(* CoDeSys 2.3 export: FILEHANDLING.EXP *)
(* Libraries: 05_Utilities\MPLCUtilities.lib 30.1.17 00:00:00, 11_System\SysLibFileAsync.lib 27.1.17 13:50:06, 11_System\SysLibProjectInfo.lib 27.1.17 13:50:06, 11_System\SysLibRtc.lib 27.1.17 13:50:06, 12_Additional\Util.lib 27.1.17 13:50:06, Internal\MPLCIntern_Utilities.lib 30.1.17 00:00:00 *)

(* Data type in CodeSamples/FileHandling *)
TYPE ST_CSVData :
STRUCT
	(********************)
	TimeStamp		: STRING(25)	:='                      ';	(* Time stamp *)
	Separator1		: BYTE			:= 16#3B; 			(* Semicolon *)
	Description1		: STRING(25)	:='                         ';	(* Description of the log data *)
	Separator2		: BYTE			:= 16#3B; 			(* Semicolon *)
	Value1				: STRING(25)	:='                         ';	(* Log value *)
	Separator3		: BYTE			:= 16#3B; 			(* Semicolon *)

	(********************)
	Description2		: STRING(25)	:='                         ';	(* Description of the log data *)
	Separato4		: BYTE				:= 16#3B; 			(* Semicolon *)
	Value2				: STRING(25)	:='                         ';	(* Log value *)
	Separator5		: BYTE			:= 16#3B; 			(* Semicolon *)
	GAP			: STRING(2)	:='  '; (*See Description*)
	CRLF3				: WORD		:= 16#0D0A;		(*Carriage return , Line feed*)

	
	(*Attention: 
	  The total number of bytes of the structure must be integer divisible by 4.
	  Use the GAP variable to compensate the size of the structure.
          !!!! STRING(25) has 26 Byte !!!
	*)

END_STRUCT
END_TYPE

(* POU CodeSamples/FileHandling/PRG_FileHandling_WriteCSVFormatedFile, FBD *)
(************************************************************************************
*
*                 Code sample  " PRG_FileHandling_WriteCSVFormatedFile "                 
*
*************************************************************************************
*
* (c) 2009 by SEW-EURODRIVE GmbH & Co KG
*
************************************************************************************
************************************************************************************
*
* PRG_FileHandling_WriteCSVFormatedFile
*
* This code sample demonstrates, how to format data into 
* CSV (comma separated values) format and write the data to SD card.
* you can use this sample program to store log data, process values ... 
* on the SD card.
* 
* Format of the file : 
*
*        2009-09-04-11:31:50 ;	Actual Speed ;	1000 ;    Actual Position ;  4096;
*        2009-09-04-11:34:13 ;   Actual Speed ;   500 ;    Actual Position ;  4096;
*
* Remark:
* If the the string values are larger than 25 characters, you have to adjust the 
* functions within the Common folder.
*
************************************************************************************)
PROGRAM PRG_FileHandling_WriteCSVFormatedFile
VAR
	(*Control *)
	bSetRtc				: BOOL;							(* Set the real time clock*)
	dtDateTimeToSet		: DT;								(* Date time to set *)
	bWriteFile				: BOOL;							(* Write data struct to SD card *)
	FileName				: STRING(25) := 'LogFile1.txt';		(* File name *)

	(* Data struct to write *)
	aCSVData	:ARRAY[1..100] OF ST_CSVData;

	(* Variables *)
	fbMC_FileHandling: MC_FileHandling;
	Mode: MC_MODE_FILEHANDLING_DM;
	fbMC_RTCManager: MPLC_RealTimeClockManager;
	dtActDateTime: DT;

END_VAR
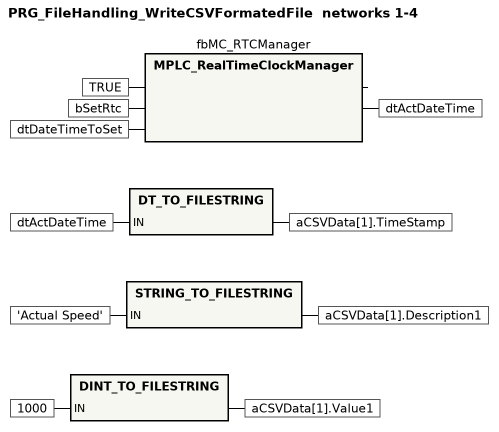
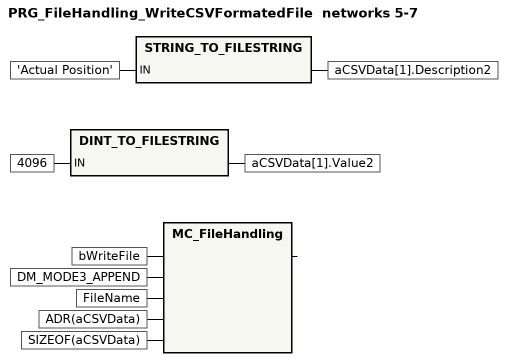
_FBD_ (* Function Block Diagram *)
NETWORK 1
	fbMC_RTCManager:MPLC_RealTimeClockManager(TRUE, bSetRtc, dtDateTimeToSet, out 2 => dtActDateTime)
NETWORK 2
	DT_TO_FILESTRING(IN: dtActDateTime) => aCSVData[1].TimeStamp
NETWORK 3
	STRING_TO_FILESTRING(IN: 'Actual Speed') => aCSVData[1].Description1
NETWORK 4
	DINT_TO_FILESTRING(IN: 1000) => aCSVData[1].Value1
NETWORK 5
	STRING_TO_FILESTRING(IN: 'Actual Position') => aCSVData[1].Description2
NETWORK 6
	DINT_TO_FILESTRING(IN: 4096) => aCSVData[1].Value2
NETWORK 7
	MC_FileHandling(bWriteFile, DM_MODE3_APPEND, FileName, ADR(aCSVData), SIZEOF(aCSVData))
_END_FBD_
(* the same logic as Structured Text *)
(* Network 1: see the listing above *)
(* Network 2 *)
aCSVData[1].TimeStamp := DT_TO_FILESTRING(IN := dtActDateTime);
(* Network 3 *)
aCSVData[1].Description1 := STRING_TO_FILESTRING(IN := 'Actual Speed');
(* Network 4 *)
aCSVData[1].Value1 := DINT_TO_FILESTRING(IN := 1000);
(* Network 5 *)
aCSVData[1].Description2 := STRING_TO_FILESTRING(IN := 'Actual Position');
(* Network 6 *)
aCSVData[1].Value2 := DINT_TO_FILESTRING(IN := 4096);
(* Network 7 *)
MC_FileHandling(bWriteFile, DM_MODE3_APPEND, FileName, ADR(aCSVData), SIZEOF(aCSVData));
END_PROGRAM

(* POU CodeSamples/FileHandling/Common/DT_TO_FILESTRING, ST *)
FUNCTION DT_TO_FILESTRING : STRING(25)
VAR_INPUT
	IN					: DT;
END_VAR
VAR
	temp: STRING(25);
	j: UINT;
END_VAR
temp :=  DT_TO_STRING(IN);
temp := DELETE (temp,3,1);

j := LEN(temp);

WHILE j < 25 DO
	temp := CONCAT(' ', temp);
	j := j + 1;
END_WHILE;

DT_TO_FILESTRING := temp;
END_FUNCTION

(* POU CodeSamples/FileHandling/Common/STRING_TO_FILESTRING, ST *)
FUNCTION STRING_TO_FILESTRING : STRING(25)
VAR_INPUT
	IN					: STRING(25);
END_VAR
VAR
	temp: STRING(25);
	j: UINT;
END_VAR
temp :=  IN;
j := LEN(temp);
WHILE j < 25 DO
	temp := CONCAT(' ', temp);
	j := j + 1;
END_WHILE;
STRING_TO_FILESTRING := temp;
END_FUNCTION

(* POU CodeSamples/FileHandling/Common/DINT_TO_FILESTRING, ST *)
FUNCTION DINT_TO_FILESTRING : STRING(25)
VAR_INPUT
	IN					: DINT;
END_VAR
VAR
	temp: STRING(25);
	j: UINT;
END_VAR
temp :=  DINT_TO_STRING(IN);
j := LEN(temp);
WHILE j < 25 DO
	temp := CONCAT(' ', temp);
	j := j + 1;
END_WHILE;
DINT_TO_FILESTRING := temp;
END_FUNCTION

(* POU CodeSamples/FileHandling/Common/DWORD_TO_FILESTRING, ST *)
FUNCTION DWORD_TO_FILESTRING : STRING(25)
VAR_INPUT
	IN:DWORD;
END_VAR
VAR
	temp: STRING(25);
	j: UINT;
END_VAR
temp :=  DWORD_TO_STRING(IN);
j := LEN(temp);
WHILE j < 25 DO
	temp := CONCAT(' ', temp);
	j := j + 1;
END_WHILE;
DWORD_TO_FILESTRING := temp;
END_FUNCTION
